PROGRAM PRG_DPL_Z_EPS
VAR
    bInit 		: BOOL := TRUE;
    bFullRange 	: BOOL;

    fbEPS		: FB_EPS;
    fbCheckEPS 	: FB_CheckEPS;
END_VAR

IF bInit THEN
    // Set Inital Values
    aDPL_Z_EPS[1].fBwd_Limits := -10;
    aDPL_Z_EPS[1].fFwd_Limits := 100;

    aDPL_Z_EPS[2].fBwd_Limits := 30;
    aDPL_Z_EPS[2].fFwd_Limits := 100;

    aDPL_Z_EPS[3].fBwd_Limits := 30;
    aDPL_Z_EPS[3].fFwd_Limits := 100;

    aDPL_Z_EPS[4].fBwd_Limits := 30;
    aDPL_Z_EPS[4].fFwd_Limits := 100;

    bInit := FALSE;
END_IF

fbEPS(eps:=aDPL_Z_EPS[2].stEPS);
fbEPS.setDescription('DPL X in [10,30]');
fbEPS.setBit(0, F_InRange(fDPL_X, 10, 30));

fbEPS(eps:=aDPL_Z_EPS[3].stEPS);
fbEPS.setDescription('RCC Y in [-34,10];RCC_Z in [-15,11]');
fbEPS.setBit(0, F_InRange(fRCC_Y, -34, 10));
fbEPS.setBit(1, F_InRange(fRCC_Z, -15, 11));

fbEPS(eps:=aDPL_Z_EPS[4].stEPS);
fbEPS.setDescription('RCC_Y in [-38,-34];RCC_Z in [-15,11];DPL_Y in [-1,40]');
fbEPS.setBit(0, F_InRange(fRCC_Y, -38, -34));
fbEPS.setBit(1, F_InRange(fRCC_Z, -15, 11));
fbEPS.setBit(2, F_InRange(fDPL_Y, -1, 40));

bFullRange := (NOT aDPL_Z_EPS[2].stEPS.bEPS_OK) AND (NOT aDPL_Z_EPS[3].stEPS.bEPS_OK) AND (NOT aDPL_Z_EPS[4].stEPS.bEPS_OK);

fbEPS(eps:=aDPL_Z_EPS[1].stEPS);
fbEPS.setDescription('Full Range');
fbEPS.setBit(0, bFullRange);

fbCheckEPS(stMotor:=M3, fPosition:=fDPL_Z, aEPSLimits:= aDPL_Z_EPS, refstForwardMotorEPS:=M3.stEPSForwardEnable, refstBackwardMotorEPS:= M3.stEPSBackwardEnable);

END_PROGRAM

(* stored: Version 1.1.0.1, ProductVersion 3.1.4022.18
   POU PRG_DPL_Z_EPS: Id {2c285499-0d64-4304-a814-9959d7ef4cde}, SpecialFunc None *)
